PROGRAM P009_ReadSavePersistent
VAR
	fbSave						:	FB_WritePersistentData;
	udiWriteCycle				:	UDINT;	
END_VAR

CASE (udiWriteCycle) OF
	0:
		;
	10:
		fbSave.START									:=	TRUE;
		udiWriteCycle									:=	20;
	20:
		IF (NOT fbSave.BUSY OR fbSave.ERR) THEN
			fbSave.START								:=	FALSE;
			udiWriteCycle								:=	0;	
		END_IF
END_CASE

fbSave.PORT												:=	851;
fbSave.TMOUT											:=	T#1000MS;

fbSave();

ACTION ACT_SaveRequest:
IF (udiWriteCycle = 0) THEN
	udiWriteCycle										:=	10;
END_IF
END_ACTION

END_PROGRAM

(* stored: Version 1.1.0.1, ProductVersion 3.1.4026.13, FileIdentifier 60433a6c91f8a3f31add880bfd458506585c5261, FileSignature 36806590f910b89f4b92b565a181202e093decdde488607c6b362af4d01b7a195a0ef65ba4a4fca2987f55c8f554d8608b798ceaf29211a83e3deb44299cedf379f781761aff64cff08079f09b63ffe45b911ea777b14c38003caf944caddf8de10012cb7cd176d7cd39fa3360a8cf57c6e32366f61d107b917f946eadb294a0ba9e33520f82ccc1fc8477a3ea20388b229841fe5a8edd0bf0a94b3aa6d2898eb948e4d30f4af6e866a0f65bb4ca1d44c7b17a573d40674d7a035561218611e9fa69eada5be396de20d0e1bd697114e9b0b2b62827ad1ee70df6b39a2c06320aceec50a7bda9faca75b8177bb4b6b48cfbd4a9b018b51316558a116b2ba054a9
   POU P009_ReadSavePersistent: Id {8023c54b-d81d-419e-8e6d-a225c75ff03b}, SpecialFunc None
   Action ACT_SaveRequest: Id {64b08d32-ad3d-42e9-bbc0-0ca444645f79} *)
